FUNCTION_BLOCK FB_PowerDelay
VAR_INPUT
	iPowerOnButton: BOOL;
	iServicesOnButton: BOOL; //option
	iPowerOffButton: BOOL;
	iIsStationSelected: BOOL;
	iPowerOnDelay: TIME:=T#3S; //option
	iMotionPowerOn:BOOL;
END_VAR
VAR_OUTPUT
	qPowerState: BOOL;
	qMotionPowerState:BOOL;
END_VAR
VAR
	timPowerOnDelay: TON;
	poweronTrig:R_TRIG;
END_VAR







//theme:zqmIUKoe-q0

//time delay for switching power on
timPowerOnDelay(	IN:= iPowerOnButton AND iIsStationSelected,
					PT:= iPowerOnDelay
				);

//OSR for setting state
	poweronTrig(		CLK:= timPowerOnDelay.Q);
//Power on, on pulse
IF poweronTrig.Q THEN
	qPowerState := 	TRUE;
END_IF
	

//power off
//option, remove iIsStationSelected if power off button is to turn off all stations?
IF iPowerOffButton AND iIsStationSelected THEN
	qPowerState := FALSE;
END_IF

//motion power on feedback logic
IF qPowerState AND iMotionPowerOn THEN
	qMotionPowerState := TRUE;
	ELSE
	qMotionPowerState := FALSE;
END_IF

END_FUNCTION_BLOCK

(* stored: Version 1.1.0.1, ProductVersion 3.1.4024.11
   POU FB_PowerDelay: Id {8fccab49-d700-484a-83d5-ad9ca7362ed3}, SpecialFunc None *)
